// TIA Portal V17 export
// export: Created 2022-05-07T16:38:48.7694435Z, ExportSetting WithDefaults, DisplayName Totally Integrated Automation Portal, DisplayVersion V17 Update 3, DisplayName TIA Portal Openness, DisplayVersion V17 Update 3, DisplayName TIA Portal Version Control Interface, DisplayVersion V17, DisplayName TIA Portal Test Suite Advanced, DisplayVersion V17 Update 1, DisplayName SINAMICS Startdrive Advanced, DisplayVersion V17 Update2, DisplayName SINAMICS Startdrive G130, G150, S120, S150, SINAMICS MV, S210, DisplayVersion V17 Update2, DisplayName SINAMICS Startdrive G110M, G120, G120C, G120D, G120P, G115D, DisplayVersion V17 Update2, DisplayName STEP 7 Professional, DisplayVersion V17 Update 3, DisplayName STEP 7 Safety, DisplayVersion V17, DisplayName WinCC UA Professional, DisplayVersion V17 Update 3
VAR_GLOBAL   // PLC tag table "Default tag table"
   System_Byte AT %MB1 : Byte;
   FirstScan AT %M1.0 : Bool;
   DiagStatusUpdate AT %M1.1 : Bool;
   AlwaysTRUE AT %M1.2 : Bool;
   AlwaysFALSE AT %M1.3 : Bool;
   Clock_Byte AT %MB0 : Byte;
   Clock_10Hz AT %M0.0 : Bool;
   Clock_5Hz AT %M0.1 : Bool;
   "Clock_2.5Hz" AT %M0.2 : Bool;
   Clock_2Hz AT %M0.3 : Bool;
   "Clock_1.25Hz" AT %M0.4 : Bool;
   Clock_1Hz AT %M0.5 : Bool;
   "Clock_0.625Hz" AT %M0.6 : Bool;
   "Clock_0.5Hz" AT %M0.7 : Bool;
   MR_Pulse AT %Q4.0 : Bool;
   MA_Pulse AT %Q4.1 : Bool;
   MR_Direction AT %Q0.0 : Bool;
   MRenable AT %M2.0 : Bool;
   MRReset AT %M2.1 : Bool;
   MRHalt AT %M2.2 : Bool;
   "MRJog-" AT %M2.3 : Bool;
   "MRJog+" AT %M2.4 : Bool;
   MRMoveRelative AT %M2.5 : Bool;
   MRMoveAbsolute AT %M2.6 : Bool;
   MA_Direction AT %Q0.1 : Bool;
   MRPower AT %M2.7 : Bool;
   MRVelocity AT %M3.0 : Bool;
   MREnabled AT %M3.5 : Bool;
   MRHomed AT %M3.1 : Bool;
   MRMoveAbsDone AT %M3.2 : Bool;
   MRStandstill AT %M3.3 : Bool;
   MRError AT %M3.4 : Bool;
   MRActualVelocity AT %MD4 : Real;
   MRActualPosition AT %MD8 : Real;
   MS_Direction AT %Q0.2 : Bool;
   ME_Direction AT %Q0.3 : Bool;
   MS_Pulse AT %Q4.2 : Bool;
   ME_Pulse AT %Q4.3 : Bool;
   AUTOMATICO AT %M3.6 : Bool;
   MANUALE AT %M3.7 : Bool;
   RIPRISTINO AT %M12.0 : Bool;
   PASSO_RIP_01 AT %M12.1 : Bool;
   PASSO_RIP_02 AT %M12.2 : Bool;
   PASSO_RIP_03 AT %M12.3 : Bool;
   STARTCICLO AT %M12.6 : Bool;
   PASSO_CICLO_01 AT %M12.7 : Bool;
   PASSO_CICLO_03 AT %M13.0 : Bool;
   PASSO_CICLO_02 AT %M13.1 : Bool;
   MRSpQuotaMoveRel AT %MD14 : Real;
   MRSpVelocitaMoveRel AT %MD18 : Real;
   MRSpQuotaMoveAbs AT %MD22 : Real;
   MRSpVelocitaMoveAbs AT %MD26 : Real;
   AUX_OK AT %M12.4 : Bool;
   AUX_OK_T AT %M12.5 : Bool;
   RESET_ALLARMI AT %M13.2 : Bool;
   MR_MAN_RELATIVE AT %M13.3 : Bool;
   MR_MAN_ABSOLUTE AT %M13.4 : Bool;
   MR_MAN_HALT AT %M13.5 : Bool;
   MS_MAN_HALT AT %M13.6 : Bool;
   MS_MAN_RELATIVE AT %M13.7 : Bool;
   MS_MAN_ABSOLUTE AT %M30.0 : Bool;
   MA_MAN_HALT AT %M30.1 : Bool;
   MA_MAN_RELATIVE AT %M30.2 : Bool;
   MA_MAN_ABSOLUTE AT %M30.3 : Bool;
   ME_MAN_HALT AT %M30.4 : Bool;
   ME_MAN_RELATIVE AT %M30.5 : Bool;
   ME_MAN_ABSOLUTE AT %M30.6 : Bool;
   "E0.0 FC HOMING MS" AT %I0.0 : Bool;
   ALLA_01_FC_HOMING_MS AT %M30.7 : Bool;
   PASSO_PASSO AT %M31.0 : Bool;
   RIPRISTINATO AT %M31.1 : Bool;
   "E0.1 FC HOMING MR" AT %I0.1 : Bool;
   ALLA_02_FC_HOMING_MR AT %M31.2 : Bool;
END_VAR
